{attribute 'qualified_only'}
{attribute 'strict'}
TYPE eGridFormingMode:
(
	Island := 0,
	Droop := 1
);
END_TYPE

(* stored: Version 1.1.0.1, ProductVersion 3.1.4026.18
   DUT eGridFormingMode: Id {f2413005-2c4b-4667-a63e-2281c616af23} *)
